// TwinCAT 3 PLC project TcAbbLinkin
// ProgramVersion: 3.1.4024.0
// libraries:
//   Tc2_Standard, * (Beckhoff Automation GmbH)
//   Tc2_System, * (Beckhoff Automation GmbH)
//   Tc3_IotBase, * (Beckhoff Automation GmbH)
//   Tc3_Module, * (Beckhoff Automation GmbH)
// project tree:
//   DUTs/ AbbLinkinConnectionConfig_Typ.TcDUT (not stored), ABBLINKIN_RWS_API_VERSION.TcDUT (not stored)
//   / PlcTask.TcTTO (not stored)
//   POUs/ MAIN.TcPOU, TcAbbLinkin.TcPOU (not stored)

// ---- POUs/MAIN.TcPOU
PROGRAM MAIN
VAR
	myRobotLink		: TcAbbLinkin;
END_VAR

END_PROGRAM
